FUNCTION_BLOCK FB_Arbiter
VAR
END_VAR

END_FUNCTION_BLOCK

(* stored: Version 1.1.0.1, ProductVersion 3.1.4022.12
   POU FB_Arbiter: Id {2ce7d585-4957-4408-a2cb-de55723dff03}, SpecialFunc None *)
